// p_ReactiveEnergy_IntoLoad
	arPM[LV01].p_ReactiveEnergy_IntoLoad := 4348107.776;
	arPM[DB_PR1_1].p_ReactiveEnergy_IntoLoad := 9371653.523;
	arPM[DB1].p_ReactiveEnergy_IntoLoad := 0;
	arPM[DB2].p_ReactiveEnergy_IntoLoad := 1578355.8;
	arPM[DB3].p_ReactiveEnergy_IntoLoad := 1391290.1;
	arPM[DB4].p_ReactiveEnergy_IntoLoad := 1935924.3;
	arPM[DB1_1].p_ReactiveEnergy_IntoLoad := 0;
	arPM[DB2_1].p_ReactiveEnergy_IntoLoad := 594440.661;
	arPM[DB3_1].p_ReactiveEnergy_IntoLoad := -0.001;
	arPM[DB4_1].p_ReactiveEnergy_IntoLoad := 889429.136;
	arPM[DB5].p_ReactiveEnergy_IntoLoad := 0;
	arPM[DB6].p_ReactiveEnergy_IntoLoad := 0;
	arPM[DB7].p_ReactiveEnergy_IntoLoad := 0;
	arPM[DB_MR].p_ReactiveEnergy_IntoLoad := 1745934.3;
	arPM[DB5_1].p_ReactiveEnergy_IntoLoad := 0;
	arPM[DB6_1].p_ReactiveEnergy_IntoLoad := 0;
	arPM[DB7_1].p_ReactiveEnergy_IntoLoad := 0;
	arPM[LV02].p_ReactiveEnergy_IntoLoad := 5022180.352;
	arPM[DB_PR1_2].p_ReactiveEnergy_IntoLoad := 5052467.319;
	arPM[DB_AIRCOMP].p_ReactiveEnergy_IntoLoad := 3158507.616;
	arPM[DB_AHU].p_ReactiveEnergy_IntoLoad := 2147945.1;
	arPM[DB8].p_ReactiveEnergy_IntoLoad := 0;
	arPM[DB9].p_ReactiveEnergy_IntoLoad := 0;
	arPM[DB10].p_ReactiveEnergy_IntoLoad := 0;
	arPM[DB8_1].p_ReactiveEnergy_IntoLoad := 0;
	arPM[DB9_1].p_ReactiveEnergy_IntoLoad := 0;
	arPM[DB10_1].p_ReactiveEnergy_IntoLoad := 0;
	arPM[A1].p_ReactiveEnergy_IntoLoad := 242355.492;
	arPM[A2].p_ReactiveEnergy_IntoLoad := 331841.589;
	arPM[A3].p_ReactiveEnergy_IntoLoad := 116816.749;
	arPM[A4].p_ReactiveEnergy_IntoLoad := -0.001;
	arPM[A5].p_ReactiveEnergy_IntoLoad := -0.001;
	arPM[LP_PR1A].p_ReactiveEnergy_IntoLoad := 0;
	arPM[LP_PR1B].p_ReactiveEnergy_IntoLoad := 0;
	arPM[LP_PR2A].p_ReactiveEnergy_IntoLoad := 0;
	arPM[LP_PR2B].p_ReactiveEnergy_IntoLoad := 0;
	arPM[LP_PR3A].p_ReactiveEnergy_IntoLoad := 0;
	arPM[DB_WH].p_ReactiveEnergy_IntoLoad := 1923034.4;
	arPM[LP_PR3B].p_ReactiveEnergy_IntoLoad := 0;
	arPM[LP_PR4A ].p_ReactiveEnergy_IntoLoad := -0.001;
	arPM[LP_PR4B].p_ReactiveEnergy_IntoLoad := -0.001;
	arPM[LP_BM].p_ReactiveEnergy_IntoLoad := 69025.3;
	arPM[DB_BM].p_ReactiveEnergy_IntoLoad := 354015.9;
	arPM[LV03].p_ReactiveEnergy_IntoLoad := 3017196.544;
	arPM[DB_MVAC1].p_ReactiveEnergy_IntoLoad := 3313250.899;
	arPM[DB_MVAC2].p_ReactiveEnergy_IntoLoad := 1470224.327;
	arPM[DB_OFF2].p_ReactiveEnergy_IntoLoad := 675362;
	arPM[LP_EL1].p_ReactiveEnergy_IntoLoad := 1784.744;
	arPM[LP_EL2].p_ReactiveEnergy_IntoLoad := 304074.4;
	arPM[DB_OFF1].p_ReactiveEnergy_IntoLoad := 808687.1;
	arPM[DB_KIT].p_ReactiveEnergy_IntoLoad := 743740.1;
	arPM[LP_WH2].p_ReactiveEnergy_IntoLoad := 868033.533;
	arPM[LP_WH1].p_ReactiveEnergy_IntoLoad := 1928.061;
	arPM[CH4].p_ReactiveEnergy_IntoLoad := 156911.535;
	arPM[CH5].p_ReactiveEnergy_IntoLoad := 106493.719;
	arPM[CH6].p_ReactiveEnergy_IntoLoad := 154188.976;
	arPM[LV04].p_ReactiveEnergy_IntoLoad := 1347330.688;
	arPM[DB_PR2].p_ReactiveEnergy_IntoLoad := 14994240.4;
	arPM[DB11].p_ReactiveEnergy_IntoLoad := 776439.1;
	arPM[DB12].p_ReactiveEnergy_IntoLoad := 2161107.6;
	arPM[DB13].p_ReactiveEnergy_IntoLoad := 2181983.7;
	arPM[DB14].p_ReactiveEnergy_IntoLoad := 4755275;
	arPM[DB11_1].p_ReactiveEnergy_IntoLoad := 163954.07;
	arPM[DB12_1].p_ReactiveEnergy_IntoLoad := 155272.319;
	arPM[DB13_1].p_ReactiveEnergy_IntoLoad := 1293062.341;
	arPM[DB14_1].p_ReactiveEnergy_IntoLoad := 4078085.288;
	arPM[DB15].p_ReactiveEnergy_IntoLoad := 4564234.1;
	arPM[DB15_1].p_ReactiveEnergy_IntoLoad := 3852128.895;
	arPM[LP_PR5A].p_ReactiveEnergy_IntoLoad := 56928.489;
	arPM[LP_PR5B].p_ReactiveEnergy_IntoLoad := 4988.717;
	arPM[LP_PR6A].p_ReactiveEnergy_IntoLoad := 4737.807;
	arPM[LP_PR6B].p_ReactiveEnergy_IntoLoad := 723.341;
// p_ReactiveEnergy_OutLoad
	arPM[LV01].p_ReactiveEnergy_OutLoad := 6873.314;
	arPM[DB_PR1_1].p_ReactiveEnergy_OutLoad := 7541.118;
	arPM[DB1].p_ReactiveEnergy_OutLoad := -88888888.4444;
	arPM[DB2].p_ReactiveEnergy_OutLoad := -88888888.4444;
	arPM[DB3].p_ReactiveEnergy_OutLoad := -88888888.4444;
	arPM[DB4].p_ReactiveEnergy_OutLoad := -88888888.4444;
	arPM[DB1_1].p_ReactiveEnergy_OutLoad := 0;
	arPM[DB2_1].p_ReactiveEnergy_OutLoad := -0.001;
	arPM[DB3_1].p_ReactiveEnergy_OutLoad := -0.001;
	arPM[DB4_1].p_ReactiveEnergy_OutLoad := -0.001;
	arPM[DB5].p_ReactiveEnergy_OutLoad := -88888888.4444;
	arPM[DB6].p_ReactiveEnergy_OutLoad := -88888888.4444;
	arPM[DB7].p_ReactiveEnergy_OutLoad := -88888888.4444;
	arPM[DB_MR].p_ReactiveEnergy_OutLoad := -88888888.4444;
	arPM[DB5_1].p_ReactiveEnergy_OutLoad := 0;
	arPM[DB6_1].p_ReactiveEnergy_OutLoad := 0;
	arPM[DB7_1].p_ReactiveEnergy_OutLoad := 0;
	arPM[LV02].p_ReactiveEnergy_OutLoad := 9729.96;
	arPM[DB_PR1_2].p_ReactiveEnergy_OutLoad := 11119.27;
	arPM[DB_AIRCOMP].p_ReactiveEnergy_OutLoad := 24.853;
	arPM[DB_AHU].p_ReactiveEnergy_OutLoad := -88888888.4444;
	arPM[DB8].p_ReactiveEnergy_OutLoad := -88888888.4444;
	arPM[DB9].p_ReactiveEnergy_OutLoad := -88888888.4444;
	arPM[DB10].p_ReactiveEnergy_OutLoad := -88888888.4444;
	arPM[DB8_1].p_ReactiveEnergy_OutLoad := 0;
	arPM[DB9_1].p_ReactiveEnergy_OutLoad := 0;
	arPM[DB10_1].p_ReactiveEnergy_OutLoad := 0;
	arPM[A1].p_ReactiveEnergy_OutLoad := 0;
	arPM[A2].p_ReactiveEnergy_OutLoad := 0;
	arPM[A3].p_ReactiveEnergy_OutLoad := 184.122;
	arPM[A4].p_ReactiveEnergy_OutLoad := 49.898;
	arPM[A5].p_ReactiveEnergy_OutLoad := 206.65;
	arPM[LP_PR1A].p_ReactiveEnergy_OutLoad := 0;
	arPM[LP_PR1B].p_ReactiveEnergy_OutLoad := 0;
	arPM[LP_PR2A].p_ReactiveEnergy_OutLoad := 0;
	arPM[LP_PR2B].p_ReactiveEnergy_OutLoad := 0;
	arPM[LP_PR3A].p_ReactiveEnergy_OutLoad := 0;
	arPM[DB_WH].p_ReactiveEnergy_OutLoad := -88888888.4444;
	arPM[LP_PR3B].p_ReactiveEnergy_OutLoad := 0;
	arPM[LP_PR4A ].p_ReactiveEnergy_OutLoad := 212934.039;
	arPM[LP_PR4B].p_ReactiveEnergy_OutLoad := -0.001;
	arPM[LP_BM].p_ReactiveEnergy_OutLoad := -88888888.4444;
	arPM[DB_BM].p_ReactiveEnergy_OutLoad := -88888888.4444;
	arPM[LV03].p_ReactiveEnergy_OutLoad := 25920.378;
	arPM[DB_MVAC1].p_ReactiveEnergy_OutLoad := 27.906;
	arPM[DB_MVAC2].p_ReactiveEnergy_OutLoad := 785.01;
	arPM[DB_OFF2].p_ReactiveEnergy_OutLoad := -88888888.4444;
	arPM[LP_EL1].p_ReactiveEnergy_OutLoad := 32356.372;
	arPM[LP_EL2].p_ReactiveEnergy_OutLoad := -88888888.4444;
	arPM[DB_OFF1].p_ReactiveEnergy_OutLoad := -88888888.4444;
	arPM[DB_KIT].p_ReactiveEnergy_OutLoad := -88888888.4444;
	arPM[LP_WH2].p_ReactiveEnergy_OutLoad := 7123.4;
	arPM[LP_WH1].p_ReactiveEnergy_OutLoad := 11322.61;
	arPM[CH4].p_ReactiveEnergy_OutLoad := 0.004;
	arPM[CH5].p_ReactiveEnergy_OutLoad := 0;
	arPM[CH6].p_ReactiveEnergy_OutLoad := 0;
	arPM[LV04].p_ReactiveEnergy_OutLoad := 4383.502;
	arPM[DB_PR2].p_ReactiveEnergy_OutLoad := -88888888.4444;
	arPM[DB11].p_ReactiveEnergy_OutLoad := -88888888.4444;
	arPM[DB12].p_ReactiveEnergy_OutLoad := -88888888.4444;
	arPM[DB13].p_ReactiveEnergy_OutLoad := -88888888.4444;
	arPM[DB14].p_ReactiveEnergy_OutLoad := -88888888.4444;
	arPM[DB11_1].p_ReactiveEnergy_OutLoad := 3757.681;
	arPM[DB12_1].p_ReactiveEnergy_OutLoad := 31580.689;
	arPM[DB13_1].p_ReactiveEnergy_OutLoad := 74213.876;
	arPM[DB14_1].p_ReactiveEnergy_OutLoad := 2244.206;
	arPM[DB15].p_ReactiveEnergy_OutLoad := -88888888.4444;
	arPM[DB15_1].p_ReactiveEnergy_OutLoad := 1914.601;
	arPM[LP_PR5A].p_ReactiveEnergy_OutLoad := 108167.521;
	arPM[LP_PR5B].p_ReactiveEnergy_OutLoad := 166369.745;
	arPM[LP_PR6A].p_ReactiveEnergy_OutLoad := 17945.167;
	arPM[LP_PR6B].p_ReactiveEnergy_OutLoad := 15140.298;
// p_Current_Avg
	arPM[LV01].p_Current_Avg := 1615.2;
	arPM[DB_PR1_1].p_Current_Avg := 1837.2587890625;
	arPM[DB1].p_Current_Avg := 71.04;
	arPM[DB2].p_Current_Avg := 77.76;
	arPM[DB3].p_Current_Avg := 126.6;
	arPM[DB4].p_Current_Avg := 322;
	arPM[DB1_1].p_Current_Avg := 37.7270994567871;
	arPM[DB2_1].p_Current_Avg := 33.3129005432129;
	arPM[DB3_1].p_Current_Avg := 57.6444261169434;
	arPM[DB4_1].p_Current_Avg := 20.1155738830566;
	arPM[DB5].p_Current_Avg := 410.8;
	arPM[DB6].p_Current_Avg := 381.8;
	arPM[DB7].p_Current_Avg := 395.76;
	arPM[DB_MR].p_Current_Avg := 0.9;
	arPM[DB5_1].p_Current_Avg := 410.8;
	arPM[DB6_1].p_Current_Avg := 381.8;
	arPM[DB7_1].p_Current_Avg := 395.76;
	arPM[LV02].p_Current_Avg := 0.9;
	arPM[DB_PR1_2].p_Current_Avg := 159.208203125;
	arPM[DB_AIRCOMP].p_Current_Avg := 251.591796875;
	arPM[DB_AHU].p_Current_Avg := 234.554837036133;
	arPM[DB8].p_Current_Avg := 147.245162963867;
	arPM[DB9].p_Current_Avg := 169.225698242187;
	arPM[DB10].p_Current_Avg := 226.534301757813;
	arPM[DB8_1].p_Current_Avg := 1768;
	arPM[DB9_1].p_Current_Avg := 848.735412597656;
	arPM[DB10_1].p_Current_Avg := 750.340087890625;
	arPM[A1].p_Current_Avg := 230.4;
	arPM[A2].p_Current_Avg := 392.64;
	arPM[A3].p_Current_Avg := 390.48;
	arPM[A4].p_Current_Avg := 112.7;
	arPM[A5].p_Current_Avg := 189.853577270508;
	arPM[LP_PR1A].p_Current_Avg := 202.786422729492;
	arPM[LP_PR1B].p_Current_Avg := 172.533237915039;
	arPM[LP_PR2A].p_Current_Avg := 217.946762084961;
	arPM[LP_PR2B].p_Current_Avg := 76.3979942321777;
	arPM[LP_PR3A].p_Current_Avg := 36.3020057678223;
	arPM[DB_WH].p_Current_Avg := 280.733093261719;
	arPM[LP_PR3B].p_Current_Avg := 0;
	arPM[LP_PR4A ].p_Current_Avg := 0.628745019435883;
	arPM[LP_PR4B].p_Current_Avg := 290.214324951172;
	arPM[LP_BM].p_Current_Avg := 169.442260742188;
	arPM[DB_BM].p_Current_Avg := 6.16329383850098;
	arPM[LV03].p_Current_Avg := 6.09428262710571;
	arPM[DB_MVAC1].p_Current_Avg := 5.7135124206543;
	arPM[DB_MVAC2].p_Current_Avg := 8.94935321807861;
	arPM[DB_OFF2].p_Current_Avg := 6.0229606628418;
	arPM[LP_EL1].p_Current_Avg := 35.4;
	arPM[LP_EL2].p_Current_Avg := 6.0403881072998;
	arPM[DB_OFF1].p_Current_Avg := 8.50614547729492;
	arPM[DB_KIT].p_Current_Avg := 8.76326274871826;
	arPM[LP_WH2].p_Current_Avg := 3.42;
	arPM[LP_WH1].p_Current_Avg := 12.64;
	arPM[CH4].p_Current_Avg := 1296;
	arPM[CH5].p_Current_Avg := 785.527038574219;
	arPM[CH6].p_Current_Avg := 380.980133056641;
	arPM[LV04].p_Current_Avg := 30.24;
	arPM[DB_PR2].p_Current_Avg := 10.6796808242798;
	arPM[DB11].p_Current_Avg := 1.52;
	arPM[DB12].p_Current_Avg := 72.8;
	arPM[DB13].p_Current_Avg := 20;
	arPM[DB14].p_Current_Avg := 64.8182525634766;
	arPM[DB11_1].p_Current_Avg := 24.2447490692139;
	arPM[DB12_1].p_Current_Avg := 14.8973999023438;
	arPM[DB13_1].p_Current_Avg := 42.1285743713379;
	arPM[DB14_1].p_Current_Avg := 115.208984375;
	arPM[DB15].p_Current_Avg := 627.2;
	arPM[DB15_1].p_Current_Avg := 497.6;
	arPM[LP_PR5A].p_Current_Avg := 68.56;
	arPM[LP_PR5B].p_Current_Avg := 47.3;
	arPM[LP_PR6A].p_Current_Avg := 120.64;
	arPM[LP_PR6B].p_Current_Avg := 140.48;
// p_PowerFactor
	arPM[LV01].p_PowerFactor := 0.955206334590912;
	arPM[DB_PR1_1].p_PowerFactor := 0.831385016441345;
	arPM[DB1].p_PowerFactor := 0.918;
	arPM[DB2].p_PowerFactor := 0.916;
	arPM[DB3].p_PowerFactor := 0.928;
	arPM[DB4].p_PowerFactor := 0.604;
	arPM[DB1_1].p_PowerFactor := 0.897019028663635;
	arPM[DB2_1].p_PowerFactor := 0.897019028663635;
	arPM[DB3_1].p_PowerFactor := 1.2460150718689;
	arPM[DB4_1].p_PowerFactor := 0.944972991943359;
	arPM[DB5].p_PowerFactor := 0.78;
	arPM[DB6].p_PowerFactor := 1.23327100276947;
	arPM[DB7].p_PowerFactor := 0.8;
	arPM[DB_MR].p_PowerFactor := 0.599858999252319;
	arPM[DB5_1].p_PowerFactor := 0.82;
	arPM[DB6_1].p_PowerFactor := 0.781;
	arPM[DB7_1].p_PowerFactor := 0.79;
	arPM[LV02].p_PowerFactor := 0.68;
	arPM[DB_PR1_2].p_PowerFactor := 0.914165019989014;
	arPM[DB_AIRCOMP].p_PowerFactor := 0.571097016334534;
	arPM[DB_AHU].p_PowerFactor := 0.948;
	arPM[DB8].p_PowerFactor := 0.943684995174408;
	arPM[DB9].p_PowerFactor := 0.947;
	arPM[DB10].p_PowerFactor := 0.616985976696014;
	arPM[DB8_1].p_PowerFactor := 0.958119094371796;
	arPM[DB9_1].p_PowerFactor := 0.85529500246048;
	arPM[DB10_1].p_PowerFactor := 0.904770016670227;
	arPM[A1].p_PowerFactor := 0.95;
	arPM[A2].p_PowerFactor := 0.779;
	arPM[A3].p_PowerFactor := 0.831;
	arPM[A4].p_PowerFactor := 0.916;
	arPM[A5].p_PowerFactor := 0.934426009654999;
	arPM[LP_PR1A].p_PowerFactor := 0.550840973854065;
	arPM[LP_PR1B].p_PowerFactor := 1.30376195907593;
	arPM[LP_PR2A].p_PowerFactor := 0.584438025951386;
	arPM[LP_PR2B].p_PowerFactor := 1.02444791793823;
	arPM[LP_PR3A].p_PowerFactor := 1.1737699508667;
	arPM[DB_WH].p_PowerFactor := 0.897457003593445;
	arPM[LP_PR3B].p_PowerFactor := 0.750712990760803;
	arPM[LP_PR4A ].p_PowerFactor := 1.02824699878693;
	arPM[LP_PR4B].p_PowerFactor := 0.87849098443985;
	arPM[LP_BM].p_PowerFactor := 0.936347007751465;
	arPM[DB_BM].p_PowerFactor := 1.16795301437378;
	arPM[LV03].p_PowerFactor := 1.26467895507813;
	arPM[DB_MVAC1].p_PowerFactor := 1.03083896636963;
	arPM[DB_MVAC2].p_PowerFactor := 1.02593994140625;
	arPM[DB_OFF2].p_PowerFactor := 1.13111698627472;
	arPM[LP_EL1].p_PowerFactor := 0.788;
	arPM[LP_EL2].p_PowerFactor := 1.08950698375702;
	arPM[DB_OFF1].p_PowerFactor := 1.02715396881104;
	arPM[DB_KIT].p_PowerFactor := 1.0314040184021;
	arPM[LP_WH2].p_PowerFactor := 1;
	arPM[LP_WH1].p_PowerFactor := 0.738;
	arPM[CH4].p_PowerFactor := 0.94951206445694;
	arPM[CH5].p_PowerFactor := 0.878521025180817;
	arPM[CH6].p_PowerFactor := 0.903286993503571;
	arPM[LV04].p_PowerFactor := 0.978;
	arPM[DB_PR2].p_PowerFactor := 1.03170502185822;
	arPM[DB11].p_PowerFactor := 0.968;
	arPM[DB12].p_PowerFactor := 0.92;
	arPM[DB13].p_PowerFactor := 0.947;
	arPM[DB14].p_PowerFactor := 0.962938010692596;
	arPM[DB11_1].p_PowerFactor := 1.01076698303223;
	arPM[DB12_1].p_PowerFactor := 0.723228991031647;
	arPM[DB13_1].p_PowerFactor := 1.15596497058868;
	arPM[DB14_1].p_PowerFactor := 0.879800021648407;
	arPM[DB15].p_PowerFactor := 0.954704165458679;
	arPM[DB15_1].p_PowerFactor := 0.939;
	arPM[LP_PR5A].p_PowerFactor := 0.972;
	arPM[LP_PR5B].p_PowerFactor := 0.87;
	arPM[LP_PR6A].p_PowerFactor := 0.872;
	arPM[LP_PR6B].p_PowerFactor := 0.86;
// PowerTotal
	arPM[LV01].p_Real_PowerTotal := 923.415375;
	arPM[DB_PR1_1].p_Real_PowerTotal := 994.784118652344;
	arPM[DB1].p_Real_PowerTotal := -88888888.4444;
	arPM[DB2].p_Real_PowerTotal := 56.96;
	arPM[DB3].p_Real_PowerTotal := 82.56;
	arPM[DB4].p_Real_PowerTotal := 73.4;
	arPM[DB1_1].p_Real_PowerTotal := 0;
	arPM[DB2_1].p_Real_PowerTotal := -1.5E+40;
	arPM[DB3_1].p_Real_PowerTotal := 24.2024536132813;
	arPM[DB4_1].p_Real_PowerTotal := 38.3368835449219;
	arPM[DB5].p_Real_PowerTotal := -88888888.4444;
	arPM[DB6].p_Real_PowerTotal := -88888888.4444;
	arPM[DB7].p_Real_PowerTotal := -88888888.4444;
	arPM[DB_MR].p_Real_PowerTotal := 2.46;
	arPM[DB5_1].p_Real_PowerTotal := 0;
	arPM[DB6_1].p_Real_PowerTotal := 0;
	arPM[DB7_1].p_Real_PowerTotal := 0;
	arPM[LV02].p_Real_PowerTotal := 1189.95925;
	arPM[DB_PR1_2].p_Real_PowerTotal := 419.044616699219;
	arPM[DB_AIRCOMP].p_Real_PowerTotal := 555.449096679688;
	arPM[DB_AHU].p_Real_PowerTotal := 112.56;
	arPM[DB8].p_Real_PowerTotal := -88888888.4444;
	arPM[DB9].p_Real_PowerTotal := -88888888.4444;
	arPM[DB10].p_Real_PowerTotal := -88888888.4444;
	arPM[DB8_1].p_Real_PowerTotal := 0;
	arPM[DB9_1].p_Real_PowerTotal := 0;
	arPM[DB10_1].p_Real_PowerTotal := 0;
	arPM[A1].p_Real_PowerTotal := 172.652557373047;
	arPM[A2].p_Real_PowerTotal := 0;
	arPM[A3].p_Real_PowerTotal := 94.6016159057617;
	arPM[A4].p_Real_PowerTotal := 174.430236816406;
	arPM[A5].p_Real_PowerTotal := 82.7287521362305;
	arPM[LP_PR1A].p_Real_PowerTotal := 0;
	arPM[LP_PR1B].p_Real_PowerTotal := 0;
	arPM[LP_PR2A].p_Real_PowerTotal := 0;
	arPM[LP_PR2B].p_Real_PowerTotal := 0;
	arPM[LP_PR3A].p_Real_PowerTotal := 0;
	arPM[DB_WH].p_Real_PowerTotal := 12.12;
	arPM[LP_PR3B].p_Real_PowerTotal := 0;
	arPM[LP_PR4A ].p_Real_PowerTotal := 5.65197658538818;
	arPM[LP_PR4B].p_Real_PowerTotal := 5.59657144546509;
	arPM[LP_BM].p_Real_PowerTotal := 2.232;
	arPM[DB_BM].p_Real_PowerTotal := 7.64;
	arPM[LV03].p_Real_PowerTotal := 841.93475;
	arPM[DB_MVAC1].p_Real_PowerTotal := 414.448852539063;
	arPM[DB_MVAC2].p_Real_PowerTotal := 222.387817382813;
	arPM[DB_OFF2].p_Real_PowerTotal := 69;
	arPM[LP_EL1].p_Real_PowerTotal := 1.16747641563416;
	arPM[LP_EL2].p_Real_PowerTotal := 0.64;
	arPM[DB_OFF1].p_Real_PowerTotal := 33.5;
	arPM[DB_KIT].p_Real_PowerTotal := 55.04;
	arPM[LP_WH2].p_Real_PowerTotal := 40.1052703857422;
	arPM[LP_WH1].p_Real_PowerTotal := 14.6377182006836;
	arPM[CH4].p_Real_PowerTotal := 0.31449943780899;
	arPM[CH5].p_Real_PowerTotal := 41.1178283691406;
	arPM[CH6].p_Real_PowerTotal := 64.0811004638672;
	arPM[LV04].p_Real_PowerTotal := 292.748;
	arPM[DB_PR2].p_Real_PowerTotal := 351.2;
	arPM[DB11].p_Real_PowerTotal := 16.96;
	arPM[DB12].p_Real_PowerTotal := 29.7;
	arPM[DB13].p_Real_PowerTotal := 43.84;
	arPM[DB14].p_Real_PowerTotal := 73.28;
	arPM[DB11_1].p_Real_PowerTotal := 0.0475543439388275;
	arPM[DB12_1].p_Real_PowerTotal := 9.4025993347168;
	arPM[DB13_1].p_Real_PowerTotal := 11.6781568527222;
	arPM[DB14_1].p_Real_PowerTotal := 79.4574737548828;
	arPM[DB15].p_Real_PowerTotal := 82.24;
	arPM[DB15_1].p_Real_PowerTotal := 15.1322813034058;
	arPM[LP_PR5A].p_Real_PowerTotal := 1.4235577583313;
	arPM[LP_PR5B].p_Real_PowerTotal := 5.79523944854736;
	arPM[LP_PR6A].p_Real_PowerTotal := 0.276815831661224;
	arPM[LP_PR6B].p_Real_PowerTotal := 0.194700807332993;
	arPM[LV01].p_Real_PowerTotal := 923.415375;
	arPM[DB_PR1_1].p_Real_PowerTotal := 994.784118652344;
	arPM[DB1].p_Real_PowerTotal := -88888888.4444;
	arPM[DB2].p_Real_PowerTotal := 56.96;
	arPM[DB3].p_Real_PowerTotal := 82.56;
	arPM[DB4].p_Real_PowerTotal := 73.4;
	arPM[DB1_1].p_Real_PowerTotal := 0;
	arPM[DB2_1].p_Real_PowerTotal := -1.5E+40;
	arPM[DB3_1].p_Real_PowerTotal := 24.2024536132813;
	arPM[DB4_1].p_Real_PowerTotal := 38.3368835449219;
	arPM[DB5].p_Real_PowerTotal := -88888888.4444;
	arPM[DB6].p_Real_PowerTotal := -88888888.4444;
	arPM[DB7].p_Real_PowerTotal := -88888888.4444;
	arPM[DB_MR].p_Real_PowerTotal := 2.46;
	arPM[DB5_1].p_Real_PowerTotal := 0;
	arPM[DB6_1].p_Real_PowerTotal := 0;
	arPM[DB7_1].p_Real_PowerTotal := 0;
	arPM[LV02].p_Real_PowerTotal := 1189.95925;
	arPM[DB_PR1_2].p_Real_PowerTotal := 419.044616699219;
	arPM[DB_AIRCOMP].p_Real_PowerTotal := 555.449096679688;
	arPM[DB_AHU].p_Real_PowerTotal := 112.56;
	arPM[DB8].p_Real_PowerTotal := -88888888.4444;
	arPM[DB9].p_Real_PowerTotal := -88888888.4444;
	arPM[DB10].p_Real_PowerTotal := -88888888.4444;
	arPM[DB8_1].p_Real_PowerTotal := 0;
	arPM[DB9_1].p_Real_PowerTotal := 0;
	arPM[DB10_1].p_Real_PowerTotal := 0;
	arPM[A1].p_Real_PowerTotal := 172.652557373047;
	arPM[A2].p_Real_PowerTotal := 0;
	arPM[A3].p_Real_PowerTotal := 94.6016159057617;
	arPM[A4].p_Real_PowerTotal := 174.430236816406;
	arPM[A5].p_Real_PowerTotal := 82.7287521362305;
	arPM[LP_PR1A].p_Real_PowerTotal := 0;
	arPM[LP_PR1B].p_Real_PowerTotal := 0;
	arPM[LP_PR2A].p_Real_PowerTotal := 0;
	arPM[LP_PR2B].p_Real_PowerTotal := 0;
	arPM[LP_PR3A].p_Real_PowerTotal := 0;
	arPM[DB_WH].p_Real_PowerTotal := 12.12;
	arPM[LP_PR3B].p_Real_PowerTotal := 0;
	arPM[LP_PR4A ].p_Real_PowerTotal := 5.65197658538818;
	arPM[LP_PR4B].p_Real_PowerTotal := 5.59657144546509;
	arPM[LP_BM].p_Real_PowerTotal := 2.232;
	arPM[DB_BM].p_Real_PowerTotal := 7.64;
	arPM[LV03].p_Real_PowerTotal := 841.93475;
	arPM[DB_MVAC1].p_Real_PowerTotal := 414.448852539063;
	arPM[DB_MVAC2].p_Real_PowerTotal := 222.387817382813;
	arPM[DB_OFF2].p_Real_PowerTotal := 69;
	arPM[LP_EL1].p_Real_PowerTotal := 1.16747641563416;
	arPM[LP_EL2].p_Real_PowerTotal := 0.64;
	arPM[DB_OFF1].p_Real_PowerTotal := 33.5;
	arPM[DB_KIT].p_Real_PowerTotal := 55.04;
	arPM[LP_WH2].p_Real_PowerTotal := 40.1052703857422;
	arPM[LP_WH1].p_Real_PowerTotal := 14.6377182006836;
	arPM[CH4].p_Real_PowerTotal := 0.31449943780899;
	arPM[CH5].p_Real_PowerTotal := 41.1178283691406;
	arPM[CH6].p_Real_PowerTotal := 64.0811004638672;
	arPM[LV04].p_Real_PowerTotal := 292.748;
	arPM[DB_PR2].p_Real_PowerTotal := 351.2;
	arPM[DB11].p_Real_PowerTotal := 16.96;
	arPM[DB12].p_Real_PowerTotal := 29.7;
	arPM[DB13].p_Real_PowerTotal := 43.84;
	arPM[DB14].p_Real_PowerTotal := 73.28;
	arPM[DB11_1].p_Real_PowerTotal := 0.0475543439388275;
	arPM[DB12_1].p_Real_PowerTotal := 9.4025993347168;
	arPM[DB13_1].p_Real_PowerTotal := 11.6781568527222;
	arPM[DB14_1].p_Real_PowerTotal := 79.4574737548828;
	arPM[DB15].p_Real_PowerTotal := 82.24;
	arPM[DB15_1].p_Real_PowerTotal := 15.1322813034058;
	arPM[LP_PR5A].p_Real_PowerTotal := 1.4235577583313;
	arPM[LP_PR5B].p_Real_PowerTotal := 5.79523944854736;
	arPM[LP_PR6A].p_Real_PowerTotal := 0.276815831661224;
	arPM[LP_PR6B].p_Real_PowerTotal := 0.194700807332993;
END_METHOD

END_PROGRAM

// ---- TEST/PGRTestFB.TcPOU
PROGRAM PGRTestFB
VAR
	Fb_Calculate : FB_CalCulateAccumulation;
	lrAccumulation : LREAL;
	CurrentTime : TIMESTRUCT;
	previoustime : TIMESTRUCT;
	bAcknowledgeNewPeriodAlarm : BOOL ;
	bMRAckAlarm	: BOOL;
	Value1Minute : LREAL;
	value1Hour	: LREAL;
	value1Day : LREAL;
	bEventHour : BOOL;
	bEventDay : BOOL;
	bFirstCycle : BOOL := TRUE;
	bReset	: BOOL;
	eTimeAccumulate : E_CompareTime;
	

END_VAR
VAR
	fbFIFO_lr : FB_FIFO_Lreal;
	bFull : BOOL;
	bempty : BOOL;
	valueOut : LREAL;
	ValueInt : LREAL;
	ackValue : BOOL;
	Addvalue : BOOL;
	ResetFIFO : BOOL;
	head : UINT;
	Tail : UINT;
	Nt_systemTime : TIMESTRUCT;
	fb_localsystemtime : TIMESTRUCT;
	
END_VAR

///
	lrAccumulation := lrAccumulation + 0.01;
	
	Fb_Calculate.TimeAccumulate := eTimeAccumulate;
	
	IF bFirstCycle THEN
		 IF Fb_Calculate.MR_Init() THEN bFirstCycle := FALSE; END_IF;
	END_IF
	
	Fb_Calculate(lrAccumulator := lrAccumulation,
					accumulatedValueOut => Value1Minute,
					previousTimestampOut => previoustime,
					bNewPeriodAlarm => bAcknowledgeNewPeriodAlarm);
					
	IF bMRAckAlarm THEN 
		IF Fb_Calculate.MR_Acknowledge() THEN
			bMRAckAlarm := FALSE ; 
		END_IF
	END_IF
	IF bReset THEN
		IF Fb_Calculate.MR_Reset() THEN
			bReset := FALSE;
		END_IF
	END_IF
/////////

bempty :=	fbFIFO_lr.IsEmpty;
bFull := fbFIFO_lr.IsFull;

IF ackValue THEN
	IF fbFIFO_lr.MR_AckGetValue() THEN
		ackValue := FALSE;
	END_IF
END_IF		

IF Addvalue THEN
	IF fbFIFO_lr.MR_AddValue( Value := ValueInt)THEN
		Addvalue := FALSE;
	END_IF
END_IF

IF ResetFIFO THEN
	IF fbFIFO_lr.MR_Reset() THEN
		ResetFIFO := FALSE;
	END_IF
END_IF
valueOut := fbFIFO_lr.OldestData;
head := fbFIFO_lr.HeadIndex;
Tail := fbFIFO_lr.TailIndex;
///
Nt_systemTime := pmDev.NT_GetTime.TIMESTR;
fb_localsystemtime := GVL.fbMachineTime.systemTime;

END_PROGRAM
